// LS Electric XG5000 project: 0122 시퀀스프로그램 편솔
// PLC LSPLC

PROGRAM NewProgram (task: 스캔 프로그램)

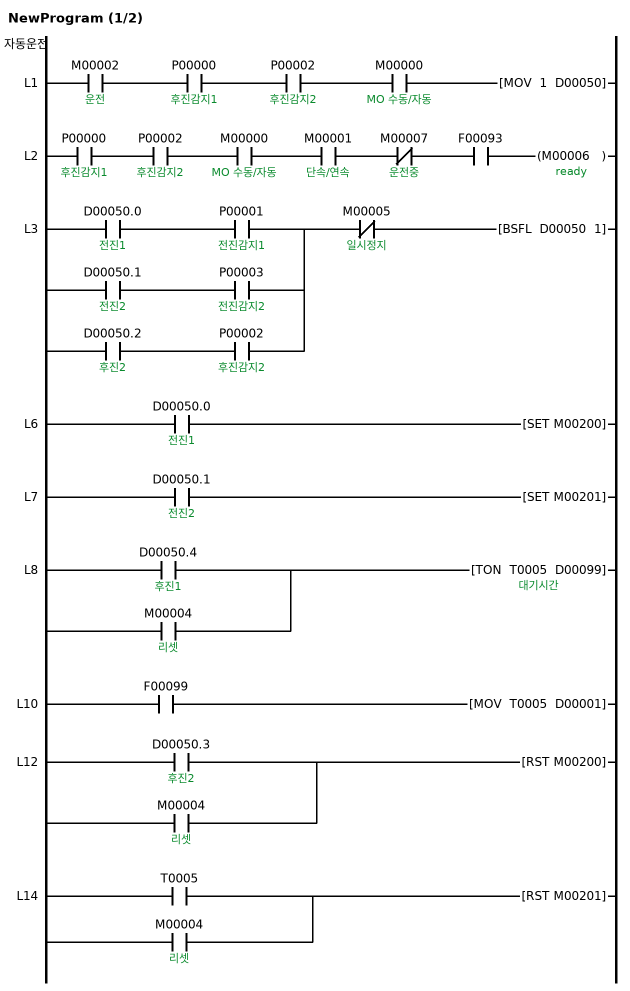
자동운전:
; L1
LOAD      M00002	// 운전
AND       P00000	// 후진감지1
AND       P00002	// 후진감지2
AND       M00000	// MO 수동/자동
MOV       1 D00050
; L2
LOAD      P00000	// 후진감지1
AND       P00002	// 후진감지2
AND       M00000	// MO 수동/자동
AND       M00001	// 단속/연속
AND NOT   M00007	// 운전중
AND       F00093
OUT       M00006	// ready
; L3
LOAD      D00050.0	// 전진1
AND       P00001	// 전진감지1
LOAD      D00050.1	// 전진2
AND       P00003	// 전진감지2
OR LOAD
LOAD      D00050.2	// 후진2
AND       P00002	// 후진감지2
OR LOAD
AND NOT   M00005	// 일시정지
BSFL      D00050 1
; L6
LOAD      D00050.0	// 전진1
SET       M00200
; L7
LOAD      D00050.1	// 전진2
SET       M00201
; L8
LOAD      D00050.4	// 후진1
OR        M00004	// 리셋
TON       T0005 D00099	// 대기시간
; L10
LOAD      F00099
MOV       T0005 D00001
; L12
LOAD      D00050.3	// 후진2
OR        M00004	// 리셋
RST       M00200
; L14
LOAD      T0005
OR        M00004	// 리셋
RST       M00201

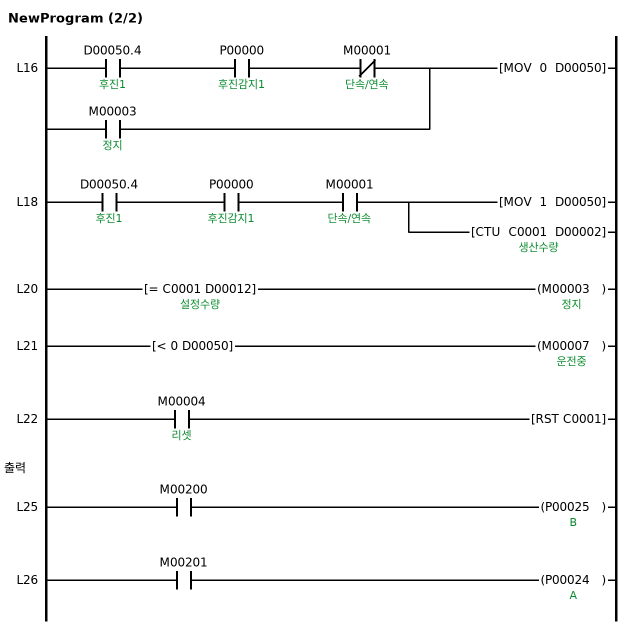
; L16
LOAD      D00050.4	// 후진1
AND       P00000	// 후진감지1
AND NOT   M00001	// 단속/연속
OR        M00003	// 정지
MOV       0 D00050
; L18
LOAD      D00050.4	// 후진1
AND       P00000	// 후진감지1
AND       M00001	// 단속/연속
MOV       1 D00050
CTU       C0001 D00002	// 생산수량
; L20
LOAD=     C0001 D00012	// 설정수량
OUT       M00003	// 정지
; L21
LOAD<     0 D00050
OUT       M00007	// 운전중
; L22
LOAD      M00004	// 리셋
RST       C0001
출력:
; L25
LOAD      M00200
OUT       P00025	// B
; L26
LOAD      M00201
OUT       P00024	// A

VARIABLES AND COMMENTS (devices not used above)
M00040	BIT	운전
M00041	BIT	NEXT
M00042	BIT	RESET
D00040.0	BIT	전진1
P00020	BIT	전진1
D00040.1	BIT	전진2
P00022	BIT	전진2
P00023	BIT	후진2
D00040.2	BIT	후진2
D00040.3	BIT	후진1